{attribute addProperty BoxType "EL3204-0162-0016"}
{attribute addProperty Id "StatusAT %I*Status_C6F82E6F1621ValueAT %I*INT16217"}
{attribute addProperty CRC "1466166969"}
{attribute addProperty SizeInBites "32"}
{attribute addProperty SizeInBytes "4"}
TYPE AI_Standard_Channel_5763EEB9 :
STRUCT
	{attribute addProperty Name "Status"}
	Status AT %I* : Status_C6F82E6F;
	{attribute addProperty Name "Value"}
	Value AT %I* : INT;
END_STRUCT
END_TYPE

(* stored: Version 1.2.0.0, ProductVersion 3.1.4024.9
   DUT AI_Standard_Channel_5763EEB9: Id {b7b65007-30a8-4f76-b308-7d10ebd0a011} *)
